{attribute addProperty BoxType "EJ5151-0000-0016"}
{attribute addProperty Id "StatusAT %I*Status_BAC5C70E1621Counter_valueAT %I*UINT16217Latch_valueAT %I*UINT16218"}
{attribute addProperty CRC "2036154"}
{attribute addProperty SizeInBites "48"}
{attribute addProperty SizeInBytes "6"}
TYPE ENC_Inputs_001F11BA :
STRUCT
	{attribute addProperty Name "Status"}
	Status AT %I* : Status_BAC5C70E;
	{attribute addProperty Name "Counter_value"}
	Counter_value AT %I* : UINT;
	{attribute addProperty Name "Latch_value"}
	Latch_value AT %I* : UINT;
END_STRUCT
END_TYPE

(* stored: Version 1.2.0.0, ProductVersion 3.1.4024.9
   DUT ENC_Inputs_001F11BA: Id {351f5e2f-f944-4195-a675-40b76e51c952} *)
